(* This function block implements the MKS392 gauge*)
FUNCTION_BLOCK FB_MKS392
VAR_INPUT
END_VAR
VAR_OUTPUT
    {attribute 'pytmc' := '
    pv:
    '}
    PG : ST_VG;
END_VAR
VAR
    rV : REAL;	// input voltage
    iTermBits: UINT := 32767 ; // The terminal's maximum value in bits
    (*IO*)
    i_iPRESS_R AT%I* :INT; // input Pressure // Link to analog Input
END_VAR

(* Real-value calculation *)
rV := 10*INT_TO_REAL(PG.i_iPRESS_R)/iTermBits;
PG.rPRESS := (LREAL_TO_REAL(EXPT(10,(2*rV)-11)));


(* Pressure gauge State checks *)

IF rV >= 0.5 AND rV <= 3.5 THEN
    PG.eState := ValidLo; //LO
ELSIF rV > 3.5 AND rV<= 6.5 THEN
    PG.eState := ValidHi; //HIGH
ELSIF rV < 0.5 THEN
    PG.eState := GaugeDisconnected; //not on
ELSE
    PG.eState := PressInvalid; //other fault - could be no gauge, controller powering up etc
END_IF



(* Pressure gauge OK checks *)
PG.xPRESS_OK := (rV <=6.5 ) AND (rV>=0.5);


(* Setpoint evaluation *)
PG.xAT_VAC := PG.xPRESS_OK AND PG.rPRESS < PG.rVAC_SP;


(*Soft IO Linking*)
ACT_IO();

ACTION ACT_IO:
PG.i_iPRESS_R :=i_iPRESS_R;
END_ACTION

METHOD M_SetBits : BOOL
VAR_INPUT
    TermBits : UINT; // The terminal's maximum value in bits
END_VAR
This^.iTermBits := TermBits;
END_METHOD

END_FUNCTION_BLOCK

(* stored: Version 1.1.0.1
   POU FB_MKS392: Id {afeb32df-f2b5-4c42-9623-5607aedfb59f}, SpecialFunc None
   Action ACT_IO: Id {593d1512-dea6-4556-9477-b1ad19e7c087}
   Method M_SetBits: Id {106bbbc2-0b06-42f6-904e-df5a4040a1c2} *)
